{attribute 'qualified_only'}
{attribute 'strict'}
TYPE nHP_Axis_ConnectionModes :
(
	None := 0,
	FitByABS := 1,
	FitByDRM := 2,
	FitByForce := 3
	
);
END_TYPE

(* stored: Version 1.1.0.1, ProductVersion 3.1.4024.12
   EnumerationTextList nHP_Axis_ConnectionModes: Id {c726e8a5-2102-421a-a540-61b05819599d} *)
